FUNCTION_BLOCK FB92
TITLE = 'pilot_Z2EV1VAD'
AUTHOR : CB

VAR
	Z2EV1ACT : FB80;
END_VAR


BEGIN


NETWORK
TITLE =
//
//	pilot/pilot_Z2/pilot_Z2EV1VAD/Z2EV1ACT
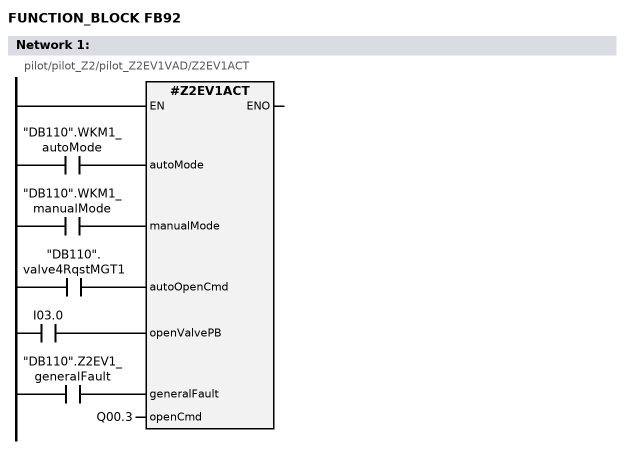
A	"DB110".WKM1_autoMode;
=	L	0.0;
BLD	103;
A	"DB110".WKM1_manualMode;
=	L	0.1;
BLD	103;
A	"DB110".valve4RqstMGT1;
=	L	0.2;
BLD	103;
A	I03.0;
=	L	0.3;
BLD	103;
A	"DB110".Z2EV1_generalFault;
=	L	0.4;
BLD	103;
CALL #Z2EV1ACT(
	autoMode := L	0.0,
	manualMode := L	0.1,
	autoOpenCmd := L	0.2,
	openValvePB := L	0.3,
	generalFault := L	0.4,
	openCmd := Q00.3
);
NOP 0;




END_FUNCTION_BLOCK
